(* PLC project P1AM Function Blocks, OpenPLC P1AM Function Blocks Library 1.0, author Thiago Alves *)
(* stored: creationDateTime 2021-11-11T02:33:11, modificationDateTime 2021-11-11T02:33:11 *)

(* Set internal RTC for Samd21 devices. If SUCCESS is zero, an error has occurred, or there aren't any modules on the bus *)
FUNCTION_BLOCK SetInternalRTC
  VAR_INPUT
    YEAR : INT;
    MONTH : INT;
    DAY : INT;
    HOUR : INT;
    MINTS : INT;
    SECONDs : INT;
  END_VAR
  VAR_OUTPUT
    DATE : DATE;
    TIME : TIME;
    SUCCESS : SINT;
  END_VAR

            SUCCESS := 0;
          
END_FUNCTION_BLOCK

(* Get internal RTC for Samd21 devices. If SUCCESS is zero, an error has occurred, or there aren't any modules on the bus *)
FUNCTION_BLOCK GetInternalRTC
  VAR_OUTPUT
    DATE : DATE;
    TIME : TIME;
    YEAR : INT;
    MONTH : INT;
    DAY : INT;
    HOUR : INT;
    MINTS : INT;
    SECOND : INT;
    SUCCESS : SINT;
  END_VAR

            SUCCESS := 0;
          
END_FUNCTION_BLOCK
